FUNCTION_BLOCK FB_SaMElementUnSuspending EXTENDS FB_SaMElement
VAR
END_VAR

METHOD FB_init : BOOL
VAR_INPUT
	bInitRetains : BOOL; // if TRUE, the retain variables are initialized (warm start / cold start)
	bInCopyCode : BOOL;  // if TRUE, the instance afterwards gets moved into the copy code (online change)
END_VAR
THIS^.SetText (eLocation := E_BaseLocation.pl, wsDescription := "Odwieszanie");
THIS^.SetText (eLocation := E_BaseLocation.en, wsDescription := "Unsuspending");
THIS^.SetText (eLocation := E_BaseLocation.de, wsDescription := "Unaussetzend");
THIS^.SetName (stName := THIS^.GetTexts ());
END_METHOD

METHOD PUBLIC InvokeStateForTopElement : BOOL
VAR_INPUT
	itfTopElement		: ITF_BaseSaMStateMethod;
END_VAR
InvokeStateForTopElement	:= itfTopElement.SP_Unsuspending ();
END_METHOD

END_FUNCTION_BLOCK

(* stored: Version 1.1.0.1
   POU FB_SaMElementUnSuspending: Id {0156b1ad-d6a5-0312-05c2-5618157b154e}, SpecialFunc None
   Method FB_init: Id {fbbf6136-5fd8-04c7-25f5-5eeb1df0e630}
   Method InvokeStateForTopElement: Id {067e775d-bbac-0460-0740-a593ba9366e0} *)
